TYPE Encoder_Typ :
STRUCT
	Status :Encoder_Status_Typ;
	Ctrl:Encoder_Control_Typ;
END_STRUCT
END_TYPE

(* stored: Version 1.1.0.1, ProductVersion 3.1.4024.3
   DUT Encoder_Typ: Id {f62bb1bb-dd63-4941-a317-a8752c608010} *)
